FUNCTION funcWithReferences : INT
VAR_IN_OUT
	num : INT;
END_VAR
VAR
END_VAR

num := num+1;

END_FUNCTION

(* stored: Version 1.1.0.1, ProductVersion 3.1.4024.11
   POU funcWithReferences: Id {d7eaaa47-cac1-4e5c-a960-7bf08f5055a0}, SpecialFunc None *)
